(* IEC 61131-3 sources: ArfBotOS/Codesys-4/ArfBotOS.fbsdev/Application.iecapp^/POU, 7 files *)

(* ---- _00_Main.prg.st ---- *)
PROGRAM _00_Main
VAR
	//
    TaskInfo : POINTER TO CmpIecTask.Task_Info2;
    TaskHandle: CmpIecTask.RTS_IEC_HANDLE;
    Result: CmpIecTask.RTS_IEC_RESULT;

	// group handler for all motion fbs
	GroupHandler: FB_GroupHandler;

	// tuning
	MoveDistance: LREAL := 5.0;
	MoveRelative: ARRAY[0..5] OF MC_MoveRelative;
	EstimateDeadTime: ARRAY[0..5] OF SMC_EstimateDeadTime;
	TuneStart: ARRAY[0..5] OF BOOL;
	TraceStart: ARRAY[0..5] OF BOOL;
	TraceStop: ARRAY[0..5] OF BOOL;
	SetTuningMoveValues: BOOL:=TRUE;
	fCycleTimeMs: LREAL; (* MainTask / SoftMotion bus cycle, ms *)
	fMeasuredLagMs: ARRAY[0..5] OF LREAL;
	fEstimatedDeadTimeRaw: ARRAY[0..5] OF LREAL; (* unclamped SMC_EstimateDeadTime median *)
	fSuggestedDeadTime: ARRAY[0..5] OF LREAL; (* D in MainTask cycles, clamped to (0, 20] *)
	nDeadTimeSamples: ARRAY[0..5] OF INT;
	bDeadTimeSuggested: ARRAY[0..5] OF BOOL;
	UseSuggestedD: ARRAY[0..5] OF BOOL;
	sDeadTimeHelp: ARRAY[0..5] OF STRING(255);
	fKpPeakLag: ARRAY[0..5] OF LREAL;
	fKpCruiseLag: ARRAY[0..5] OF LREAL;
	fKpFinalLag: ARRAY[0..5] OF LREAL;
	fKpOvershoot: ARRAY[0..5] OF LREAL;
	fKpUndershoot: ARRAY[0..5] OF LREAL;
	nKpReversals: ARRAY[0..5] OF INT;
	nKpVelReversals: ARRAY[0..5] OF INT;
	fSuggestedKp: ARRAY[0..5] OF LREAL;
	bKpSuggested: ARRAY[0..5] OF BOOL;
	UseSuggestedKp: ARRAY[0..5] OF BOOL;
	RaiseKp: ARRAY[0..5] OF BOOL;
	LowerKp: ARRAY[0..5] OF BOOL;
	sKpVerdict: ARRAY[0..5] OF STRING(16);
	sKpHelp: ARRAY[0..5] OF STRING(255);

	// homing
	ProcessHome: FB_HomingProcessor;
	HomingStatusText: STRING(255);

	// jogging
	ProcessJog: FB_JogProcessor;
	JogStatusText: STRING(255);
	ButtonTextIndex: INT:=0;

	// cnc
	VisuStruct3DControl_J: VisuStruct3DControl;
	TrackPosition: FB_PositionTracker;

	// program processor
	ProcessPrograms: FB_ProgramProcessor;
	ProcessCommand_ActiveProgram: UINT := 0;
	ActiveCommandDetails: STRING(255):='';

	// controller
	Controller: FB_Controller;

	//
	EnableRtrig: R_TRIG;
	EnableFtrig: F_TRIG;
	_i, _j, _k: INT;
	BuildTests: BOOL:=FALSE;
	FirstScan: BOOL:=TRUE;

END_VAR

{region "utility"}
    (* Get the current task info *)
    {IF defined (IsSimulationMode)}
        GVL_App.dwMainInterval := 1000;
    {ELSE}
        TaskHandle := CmpIecTask.IecTaskGetCurrent(ADR(Result));
        TaskInfo := CmpIecTask.IecTaskGetInfo3(TaskHandle, ADR(Result));
        GVL_App.dwMainInterval := TaskInfo^.dwInterval;
    {END_IF}

	GVL_App.ResetRtrig(CLK:=GVL_App.Reset);
	IF GVL_App.ResetRtrig.Q THEN
		GVL_App.Reset := FALSE;
        AlarmManager.AlarmGlobals.g_AlarmHandler.AcknowledgeAll();
        //AlarmManager.AlarmGlobals.g_AlarmHandler.AcknowledgeAllOfGroup(Alm_AlarmConfiguration_Alarmgroup_IDs.ID_Processors); // only processors
	END_IF

	GVL_App.LicenseStatus();

	IF FirstScan THEN
		M_Init();
	END_IF

	IF BuildTests THEN
		BuildTests := FALSE;
		M_BuildTests();
	END_IF

	EnableRtrig(CLK:=GVL_App.PowerOn);
	EnableFtrig(CLK:=GVL_App.PowerOn);
	IF EnableRTrig.Q THEN
		GVL_App.Enable := TRUE;
	END_IF
	IF EnableFTrig.Q THEN
		GVL_App.Enable := FALSE;
	END_IF
{endregion}

{region "methods"}
	_M_GroupHandler();
    _M_Jogging();
    _M_Homing();
    _M_Cnc();
    _M_Processor();
	_M_Controller();
	_M_Tuning();
{endregion}

// do not put anything below this
FirstScan:=FALSE;
END_PROGRAM

(* ---- _10_Robot.prg.st ---- *)
PROGRAM _10_Robot
VAR
	//
	AR4Inputs: ARRAY [0..31] OF BYTE;
	AR4Outputs: ARRAY [0..31] OF BYTE;

	//
	rx_heartbeat: BOOL;
	rx_en: BOOL;
	rx_j1_limit, rx_j2_limit, rx_j3_limit: BOOL;
	rx_j4_limit, rx_j5_limit, rx_j6_limit: BOOL;

	//
	InitializeDrives: BOOL;

	//
	FirstScan: BOOL:=TRUE;

END_VAR

//
IF FirstScan THEN
	M_Init(FALSE);
END_IF

_M_Init();
_M_HandleIO();

// do not put anything below this
FirstScan := FALSE;
END_PROGRAM

(* ---- _20_Io.prg.st ---- *)
PROGRAM _20_Io
VAR
	//
	IoInputs: ARRAY [0..31] OF BYTE;
	IoOutputs: ARRAY [0..31] OF BYTE;

	//
	rx_heartbeat: BOOL;
	rx_en: BOOL;

    //
    IoOption: INT:=0;

	//
	FirstScan: BOOL:=TRUE;
END_VAR

//
IF FirstScan THEN
    //
END_IF

// leaving this pragma here for reference and for learning.
// it is not needed and was an attempt to parameterize configuring the IO
// the project define evaluates and could be a super handy technique in the future so I'll leave it here for reference.
// the defines for the project can be found in the Toolbar under Project -> Project Settings... -> Compile options -> Edit project defines...
{IF project_defined(IoOption1)}
    //IoOption := 1;
    //_M_MapIoOption1();
{ELSIF project_defined(IoOption2)}
    //IoOption := 2;
    //_M_MapIoOption2();
{ELSE}
    //IoOption := 0;
{END_IF}

// detect if the slave is connected and map its IO
IF IoOption1.wState = ETC_SLAVE_STATE.ETC_SLAVE_OPERATIONAL THEN
    _M_MapIoOption1();
END_IF
IF IoOption2.wState = ETC_SLAVE_STATE.ETC_SLAVE_OPERATIONAL THEN
    _M_MapIoOption2();
END_IF

// do not put anything below this
FirstScan := FALSE;
END_PROGRAM

(* ---- _30_Visu.prg.st ---- *)
PROGRAM _30_Visu
VAR
    // alarms
	itfAlarmConfiguration : AlarmManager.IAlarmConfiguration;
    itfAlarmConfiguration7 : AlarmManager.IAlarmConfiguration7;
    iAlarmCfg : INT;

    //
	SelectedProgramNumber: INT;
	SelectedRecipeRowIndex: INT;
    SelectedRecipeRowIndexLast: INT;
	RecipeRowSelected: BOOL;
	InsertLineAbove: BOOL;
	InsertLineBelow: BOOL;
	DeleteLine: BOOL;
	CopySelectedCommand: BOOL;
	CopiedCommandType: DUT_CommandType;
	CopiedCommandString: STRING(GVL_App.COMMAND_LEN);
	CopiedCommandComment: STRING;
	PasteCommand: BOOL;
	JumpRowChanged: BOOL;
    ScrollingBegin: BOOL;
    ScrollingSingleUp: BOOL;
    ScrollingSingleDown: BOOL;
    ScrollingPageUp: BOOL;
    ScrollingPageDown: BOOL;
    ScrollingEnd: BOOL;

	_i,_j,_k: INT;

	SetStoredPositionAsCurrent: BOOL;
	SelectedStoredPosition: UINT;
	SetVisionRegisterAsCurrent: BOOL;
	SelectedVisionRegister: UINT;
	SelectedFlag: UINT;

	//
	TeachPosition: BOOL;
	stTeachPosition: ST_MoveCmd;

	//
	MoveCmdParser: FB_ParseMoveCmd;
	stMoveCmd: ST_MoveCmd;
	MoveCmdVisu: AddMoveCmd_VISU_STRUCT;

	//
	OutputCmdParser: FB_ParseOutputCmd;
	stOutputCmd: ST_OutputCmd;
	OutputCmdVisu: AddOutputCmd_VISU_STRUCT;

	//
	PauseCmdParser: FB_ParsePauseCmd;
	stPauseCmd: ST_PauseCmd;
	PauseCmdVisu: AddPauseCmd_VISU_STRUCT;

	//
	VisionCmdParser : FB_ParseVisionCmd;
	stVisionCmd : ST_VisionCmd;
	VisionCmdVisu: AddVisionCmd_VISU_STRUCT;

	//
	VarSetCmdParser : FB_ParseVarSetCmd;
	stVarSetCmd : ST_VarSetCmd;
	VarSetCmdVisu: AddVarSetCmd_VISU_STRUCT;

	//
	CncCmdParser : FB_ParseCncCmd;
	stCncCmd : ST_CncCmd;
	CncCmdVisu: AddCncCmd_VISU_STRUCT;

	//
	LogicCmdParser : FB_ParseLogicCmd;
	stLogicCmd : ST_LogicCmd;
	LogicCmdVisu: AddLogicCmd_VISU_STRUCT;

	//
	CurrentVisu: STRING;
	OpenDialog: VU.FbOpenDialogExtended;

END_VAR

//
GVL_App.lrGripperOpen := SEL(GVL_App.CmdIO.Output[0], 0.0, 100.0);

// scrolling
IF ScrollingBegin OR ScrollingSingleUp OR ScrollingSingleDown OR ScrollingPageUp OR ScrollingPageDown OR ScrollingEnd
    AND_THEN SelectedRecipeRowIndex <> SelectedRecipeRowIndexLast THEN
        SelectedRecipeRowIndexLast := SelectedRecipeRowIndex;
        ScrollingBegin := ScrollingSingleUp := ScrollingSingleDown := ScrollingPageUp := ScrollingPageDown := ScrollingEnd := FALSE;
END_IF

//
IF (InsertLineAbove OR InsertLineBelow) AND RecipeRowSelected THEN
	//
	IF InsertLineAbove THEN
		InsertLineAbove := FALSE;
		_j := SelectedRecipeRowIndex + 1;
	ELSIF InsertLineBelow THEN
		InsertLineBelow := FALSE;
		_j := SelectedRecipeRowIndex + 2;
	END_IF
	//
	FOR _i := GVL_App.PROG_CMDS_ARR_END TO _j BY -1 DO
		// shift all data
		IF _i >= GVL_App.PROG_CMDS_ARR_BEG AND _i <= GVL_App.PROG_CMDS_ARR_END THEN // can never really be too careful am I right?
			//
			MemUtils.MemCpy(pbyDest:=ADR(PersistentVars.Programs[SelectedProgramNumber].Commands[_i]),
							pbySrc:=ADR(PersistentVars.Programs[SelectedProgramNumber].Commands[_i - 1]),
							dwSize:=SIZEOF(PersistentVars.Programs[SelectedProgramNumber].Commands[_i]));
		END_IF
	END_FOR
	FOR _k := GVL_App.PROG_CMDS_ARR_END TO GVL_App.PROG_CMDS_ARR_BEG BY -1 DO
		// check if the command is a logic command with a jump function
		// if so, we need to move the jump row automatically so it doesnt point to an invalid command.
		// otherwise, the user would have to manually change this each time they move rows.
		JumpRowChanged := F_ChangeJumpRow(Command:=PersistentVars.Programs[SelectedProgramNumber].Commands[_k], BeginningRow:= _j-1, Change:= 1);
	END_FOR
	//
	PersistentVars.Programs[SelectedProgramNumber].Commands[_j - 1].CommandType := DUT_CommandType.Disabled;
	PersistentVars.Programs[SelectedProgramNumber].Commands[_j - 1].CommandString := '';
	PersistentVars.Programs[SelectedProgramNumber].Commands[_j - 1].CommandComment := '';
END_IF

//
IF DeleteLine AND RecipeRowSelected THEN
	DeleteLine := FALSE;
	FOR _i := SelectedRecipeRowIndex TO GVL_App.PROG_CMDS_ARR_END - 1 BY 1 DO
		IF _i >= GVL_App.PROG_CMDS_ARR_BEG AND _i <= GVL_App.PROG_CMDS_ARR_END THEN // can never really be too careful am I right?
			//
			MemUtils.MemCpy(pbyDest:=ADR(PersistentVars.Programs[SelectedProgramNumber].Commands[_i]),
							pbySrc:=ADR(PersistentVars.Programs[SelectedProgramNumber].Commands[_i + 1]),
							dwSize:=SIZEOF(PersistentVars.Programs[SelectedProgramNumber].Commands[_i]));
		END_IF
	END_FOR
	FOR _k := GVL_App.PROG_CMDS_ARR_END TO GVL_App.PROG_CMDS_ARR_BEG BY -1 DO
		// check if the command is a logic command with a jump function
		// if so, we need to move the jump row automatically so it doesnt point to an invalid command.
		// otherwise, the user would have to manually change this each time they move rows.
		JumpRowChanged := F_ChangeJumpRow(Command:=PersistentVars.Programs[SelectedProgramNumber].Commands[_k], BeginningRow:= SelectedRecipeRowIndex, Change:= -1);
	END_FOR
END_IF

//
IF SetStoredPositionAsCurrent THEN
	SetStoredPositionAsCurrent := FALSE;
	PersistentVars.StoredPositions[SelectedStoredPosition].Position.X := F_RoundLreal(_00_Main.ProcessJog.Position.v[0],2);
	PersistentVars.StoredPositions[SelectedStoredPosition].Position.Y := F_RoundLreal(_00_Main.ProcessJog.Position.v[1],2);
	PersistentVars.StoredPositions[SelectedStoredPosition].Position.Z := F_RoundLreal(_00_Main.ProcessJog.Position.v[2],2);
	PersistentVars.StoredPositions[SelectedStoredPosition].Position.A := F_RoundLreal(_00_Main.ProcessJog.Position.v[3],2);
	PersistentVars.StoredPositions[SelectedStoredPosition].Position.B := F_RoundLreal(_00_Main.ProcessJog.Position.v[4],2);
	PersistentVars.StoredPositions[SelectedStoredPosition].Position.C := F_RoundLreal(_00_Main.ProcessJog.Position.v[5],2);
END_IF

//
IF TeachPosition THEN
	TeachPosition := FALSE;
	//
	stTeachPosition.MoveType := DUT_Command_MoveType.DirectMove;
	stTeachPosition.Speed := 50;
	stTeachPosition.PositionType := DUT_Command_PositionType.AbsolutePosition;
	stTeachPosition.CoordSystem := _00_Main.ProcessJog.CoordSystem;
	stTeachPosition.CoordRef.X := F_RoundLreal(_00_Main.ProcessJog.Position.v[0],2);
	stTeachPosition.CoordRef.Y := F_RoundLreal(_00_Main.ProcessJog.Position.v[1],2);
	stTeachPosition.CoordRef.Z := F_RoundLreal(_00_Main.ProcessJog.Position.v[2],2);
	stTeachPosition.CoordRef.A := F_RoundLreal(_00_Main.ProcessJog.Position.v[3],2);
	stTeachPosition.CoordRef.B := F_RoundLreal(_00_Main.ProcessJog.Position.v[4],2);
	stTeachPosition.CoordRef.C := F_RoundLreal(_00_Main.ProcessJog.Position.v[5],2);
	PersistentVars.Programs[SelectedProgramNumber].Commands[SelectedRecipeRowIndex].CommandType := DUT_CommandType.MoveCommand;
	PersistentVars.Programs[SelectedProgramNumber].Commands[SelectedRecipeRowIndex].CommandString := F_BuildMoveCmd(stTeachPosition);
	PersistentVars.Programs[SelectedProgramNumber].Commands[SelectedRecipeRowIndex].CommandComment := 'Taught position';
END_IF

//
IF PasteCommand THEN
	PasteCommand := FALSE;
	PersistentVars.Programs[SelectedProgramNumber].Commands[SelectedRecipeRowIndex].CommandType := CopiedCommandType;
	PersistentVars.Programs[SelectedProgramNumber].Commands[SelectedRecipeRowIndex].CommandString := CopiedCommandString;
	PersistentVars.Programs[SelectedProgramNumber].Commands[SelectedRecipeRowIndex].CommandComment := CopiedCommandComment;
END_IF

//
IF CopySelectedCommand THEN
	CopySelectedCommand := FALSE;

	//
	CopiedCommandType := PersistentVars.Programs[SelectedProgramNumber].Commands[SelectedRecipeRowIndex].CommandType;
	CopiedCommandString := PersistentVars.Programs[SelectedProgramNumber].Commands[SelectedRecipeRowIndex].CommandString;
	CopiedCommandComment := PersistentVars.Programs[SelectedProgramNumber].Commands[SelectedRecipeRowIndex].CommandComment;

	CASE PersistentVars.Programs[SelectedProgramNumber].Commands[SelectedRecipeRowIndex].CommandType OF
		DUT_CommandType.Disabled:
			//

		DUT_CommandType.MoveCommand:
			MoveCmdParser(Command := PersistentVars.Programs[SelectedProgramNumber].Commands[SelectedRecipeRowIndex].CommandString);
			stMoveCmd := MoveCmdParser.stCommand;

		DUT_CommandType.PauseCommand:
			PauseCmdParser(Command:=PersistentVars.Programs[SelectedProgramNumber].Commands[SelectedRecipeRowIndex].CommandString);
			stPauseCmd := PauseCmdParser.stCommand;

		DUT_CommandType.InputCommand:
			//

		DUT_CommandType.OutputCommand:
			OutputCmdParser(Command:=PersistentVars.Programs[SelectedProgramNumber].Commands[SelectedRecipeRowIndex].CommandString);
			stOutputCmd := OutputCmdParser.stCommand;

		DUT_CommandType.VisionCommand:
			VisionCmdParser(Command:=PersistentVars.Programs[SelectedProgramNumber].Commands[SelectedRecipeRowIndex].CommandString);
			stVisionCmd := VisionCmdParser.stCommand;

		DUT_CommandType.VarSetCommand:
			VarSetCmdParser(Command:=PersistentVars.Programs[SelectedProgramNumber].Commands[SelectedRecipeRowIndex].CommandString);
			stVarSetCmd := VarSetCmdParser.stCommand;

		DUT_CommandType.CncCommand:
			CncCmdParser(Command:=PersistentVars.Programs[SelectedProgramNumber].Commands[SelectedRecipeRowIndex].CommandString);
			stCncCmd := CncCmdParser.stCommand;

		DUT_CommandType.LogicCommand:
			LogicCmdParser(Command:=PersistentVars.Programs[SelectedProgramNumber].Commands[SelectedRecipeRowIndex].CommandString);
			stLogicCmd := LogicCmdParser.stCommand;

	END_CASE

END_IF

// should be called after CopySelectedCommand case statement
CurrentVisu := VisuElems.CurrentVisu;
OpenDialog(
	xExecute:= ,
	xDone=> ,
	xBusy=> ,
	xError=> ,
	itfClientFilter:= ,
	eError=> ,
	sDialogName:= ,
	xModal:= TRUE, // TRUE - visu in background cannot be used
	pTopLeftPosition:= ,
	itfDialogOpenedListener:= ,
	pbyDialogInterfaceData:= ,
	udiDialogInterfaceDataSize:= ,
	itfDialogCloseListener:= ,
	pbyTagForDialogClosed:= ,
	dwDialogFlags:= );
IF (OpenDialog.xExecute AND OpenDialog.xDone)
	OR OpenDialog.xError
	THEN
		OpenDialog.xExecute := FALSE;
END_IF

// alarms
IF GVL_App.xClearHistory THEN
    FOR iAlarmCfg := 0 TO AlarmManager.AlarmGlobals.g_AlarmHandler.AlarmConfigurationCount - 1 DO
        itfAlarmConfiguration := AlarmManager.AlarmGlobals.g_AlarmHandler.GetAlarmConfiguration(iAlarmCfg);
        IF __QUERYINTERFACE(itfAlarmConfiguration, itfAlarmConfiguration7) THEN
            itfAlarmConfiguration7.ClearHistory(xKeepActiveAlarms := TRUE); // xKeepActiveAlarms := TRUE so a live fault isn’t ripped out of the recorder.
        END_IF
    END_FOR
    GVL_App.xClearHistory := FALSE;
END_IF
END_PROGRAM

(* ---- _40_Vision.prg.st ---- *)
PROGRAM _40_Vision
// vision is separated into its own program so that we can
// assign it to its own core! how awesome is that?!
VAR
	ProcessVisionCommand: FB_VisionCmdProcessor;
   	HostName   : STRING;
	VisionSystemUrl: STRING;
	VisionOutputImageUrl: STRING;
	VisionSystemIpAddress_Last: STRING(19);
    VisionOutputImageScaling: REAL := 1000.0;
    VisionImageWidth: INT:=365; // TODO figure out a way to dynamically set this based on the values set in the visu element properties
    VisionImageHeight: INT:=255;
END_VAR
VAR CONSTANT
	LocalIpAddress: STRING(19):='127.0.0.1';
END_VAR

// used to show the output image on the HMI
// local vision:  http://<plc-hostname>.local:5000/output_sized?width=365&height=255
// remote vision: http://<vision-ip>:5000/output_sized?width=365&height=255
IF PersistentVars.VisionSystemIpAddress <> VisionSystemIpAddress_Last THEN
    VisionSystemIpAddress_Last := PersistentVars.VisionSystemIpAddress;
    //
    IF PersistentVars.VisionSystemIpAddress = LocalIpAddress THEN
        // WebVisu runs in the PC browser, so 127.0.0.1 would hit the PC.
        // Use this PLC's mDNS name instead.
        // https://forge.codesys.com/forge/talk/Runtime/thread/61d60a9fb7/
        SysSockGetHostName(szHostName:=HostName, diNameLen:=SIZEOF(HostName));
        VisionSystemUrl := CONCAT('http://', HostName);
        VisionSystemUrl := CONCAT(VisionSystemUrl, '.local');
    ELSE
        // Dedicated vision Pi: the Programming HMI IP is already that box.
        VisionSystemUrl := CONCAT('http://', PersistentVars.VisionSystemIpAddress);
    END_IF
    //
    VisionSystemUrl := CONCAT(VisionSystemUrl, ':5000/vision');
    VisionOutputImageUrl := CONCAT(VisionSystemUrl,'/output_sized?width=');
    VisionOutputImageUrl := CONCAT(VisionOutputImageUrl,INT_TO_STRING(VisionImageWidth));
    VisionOutputImageUrl := CONCAT(VisionOutputImageUrl,'&height=');
    VisionOutputImageUrl := CONCAT(VisionOutputImageUrl,INT_TO_STRING(VisionImageHeight));
END_IF

//
ProcessVisionCommand(
    VisionSystemIpAddress:= PersistentVars.VisionSystemIpAddress,
    VisionSystemPort:= PersistentVars.VisionSystemPort,
    StoredPositions:= PersistentVars.StoredPositions,
    VisionRegisters:= PersistentVars.VisionRegisters,
    Flags:= PersistentVars.Flags,
    LogicCmdIO:= GVL_App.CmdIO,
    ItfUnitMode=> ,
    Error=> ,
    ErrorDescription=> ,
    VisionStateText=> );
END_PROGRAM

(* ---- _50_Retains.prg.st ---- *)
PROGRAM _50_Retains
VAR
	//
	SaveRetain, RestoreRetain: BOOL;
	pApplication : POINTER TO CmpApp.APPLICATION;
	ResultFind, ResultStore, ResultRestore: UDINT;

	//
	FirstScan: BOOL:=TRUE;
END_VAR

IF RestoreRetain THEN
	pApplication := CmpApp.AppFindApplicationByName('Application', ADR(ResultFind));
	ResultRestore := CmpApp.AppRestoreRetainsFromFile(pApplication, './Application/BackupRetain.ret');
	RestoreRetain := FALSE;
END_IF

IF SaveRetain THEN
	pApplication := CmpApp.AppFindApplicationByName('Application', ADR(ResultFind));
    ResultStore := AppStoreRetainsInFile(pApplication, './Application/BackupRetain.ret');
   	ResultStore := AppStoreRetainsInFile(pApplication, './Application/Application.ret');
   	SaveRetain := FALSE;
END_IF

// do not put anything below this
FirstScan := FALSE;
END_PROGRAM

(* ---- _60_PathPlanner.prg.st ---- *)
PROGRAM _60_PathPlanner
VAR
	PlanPath: FB_CncPathPlanner;
END_VAR
VAR CONSTANT
	wVarCount : WORD := 1;
END_VAR
VAR
	lrR1 : LREAL:=30;

	astVar : ARRAY [0..wVarCount] OF SMC_SingleVar :=
			[(strVarName:='R1', pAdr := ADR(lrR1), eVarType := SMC_VarType.SMC_TYPE_LREAL)];

	stVarList : SMC_VarList := (wNumberVars := wVarCount, psvVarlist := ADR(astVar));
END_VAR

// this has to be called in a separate task with lower priority
// https://content.helpme-codesys.com/en/libs/SM3_CNC/Current/SM_CNC_POUs/NC2/Interpreter/SMC_NCInterpreter.html
PlanPath(VarList:= stVarList, DataOut=> );
END_PROGRAM
